FUNCTION_BLOCK "FB_ProveInner"
{ S7_Optimized_Access := 'TRUE' }
VERSION : 0.1
   VAR_INPUT
      step : Int;
   END_VAR

   VAR_OUTPUT
      count : Int;
   END_VAR


BEGIN
	// counts on from cycle to cycle: the instance keeps it
	#count := #count + #step;
END_FUNCTION_BLOCK

